ABB RobotStudio station: dual_weld_positioner.rspag

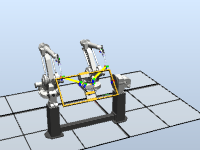
--- station ---
Station dual_weld_positioner (saved by RobotStudio 6.5.7392.129)
Controller 1410_dual_weld, task T_POS1: task frame (RAPID world) sits at (0, 0, 300) mm in the station
Controller 1410_dual_weld, task T_ROB2: task frame (RAPID world) sits at (0, 0, 300) mm in the station
Controller 1410_dual_weld, task T_ROB1: task frame (RAPID world) sits at (0, 0, 300) mm in the station
Controller 1410_dual_weld
  mechanical unit ROB_1: IRB1410_5_144__01, 6 joints, base frame (0, 0, 0) mm
  mechanical unit ROB_2: IRB1410_5_144__01_2, 6 joints, base frame (0, -1088.08, 0) mm
  mechanical unit STN1: IRBP_L300_L1250_M2009_REV1_01, 1 joints, base frame (1232.35, 0, 650) mm, rotated rx 0 ry -90 rz 90 deg
Layout (positions relative to the parent item):
  - IRB1410_5_144__01 [mechanism, from Robots\IRB1410_5_144_G_01.rslib] at (0, 0, 300) mm; joint values [0, -0.6808, -0.1899, 0, 0.7135, 0] (rad or m)
  - IRB1410_5_144__01_2 [mechanism, from Robots\IRB1410_5_144_G_01.rslib] at (0, -1088.08, 300) mm; joint values [0, -0.4622, -0.0882, 0, 0.6118, 0] (rad or m)
  - IRBP_L300_L1250_M2009_REV1_01 [mechanism] at (1232.35, 0, 0) mm; joint values [-0.7854] (rad or m)
      links: Base, Link1
  - test part [part] at (1232.35, 0, 950) mm, rotated rx 90 ry -45 rz 0 deg
  - Binzel_air_22 [mechanism, from Tools\Binzel_air_22.rslib] at (530.37, 0, 1452.5) mm, rotated rx 180 ry 60 rz 180 deg
  - Binzel_air_22_2 [mechanism, from Tools\Binzel_air_22.rslib] at (662.71, -1088.08, 1452.5) mm, rotated rx -180 ry 60 rz -180 deg
Attachment: test part is attached to IRBP_L300_L1250_M2009_REV1_01 / Link1
Attachment: Binzel_air_22 is attached to IRB1410_5_144__01 / Link6
Attachment: Binzel_air_22_2 is attached to IRB1410_5_144__01_2 / Link6

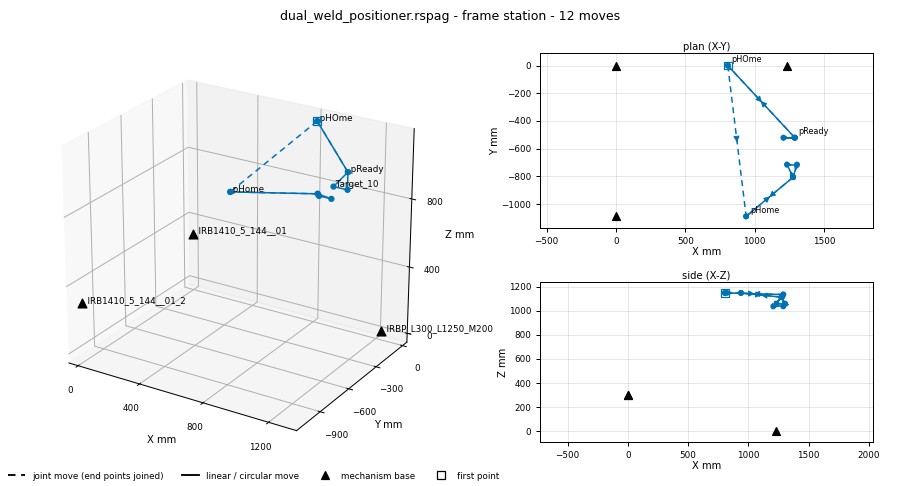
[picture p0: tool path of dual_weld_positioner.rspag in frame station, 12 of 17 moves have a stored position in this frame; points joined in program order, loops and branches not executed]
--- Backups/1410_dual_weld/RAPID/TASK1/PROGMOD/CalibData.mod ---
MODULE CalibData
	PERS tooldata tWeldGun:=[TRUE,[[125.800591275,0,391.268161315],[0.898794046,0,0.438371147,0]],[3,[0,0,100],[0,1,0,0],0,0,0]];
ENDMODULE

--- Backups/1410_dual_weld/RAPID/TASK1/PROGMOD/Module1.mod ---
MODULE Module1
    CONST robtarget pHOme:=[[806.318054074,0,847.919423179],[0.069756481,0,0.99756405,0],[0,0,0,0],[9E+09,9E+09,9E+09,9E+09,9E+09,9E+09]];
    CONST robtarget pReady:=[[1289.982978993,-520.829920074,834.561570832],[0.069756682,-0.00000004,0.997564036,-0.000000048],[-1,0,-1,0],[9E+09,9E+09,9E+09,9E+09,9E+09,9E+09]];
    CONST robtarget Target_10:=[[1207.204988688,-520.829978488,736.805052893],[0.06975661,-0.000000027,0.997564041,-0.000000051],[-1,0,-1,0],[9E+09,9E+09,9E+09,9E+09,9E+09,9E+09]];
    CONST robtarget Target_20:=[[1289.98298789,-520.829945867,736.805062664],[0.06975665,-0.000000033,0.997564038,-0.000000053],[-1,0,-1,0],[9E+09,9E+09,9E+09,9E+09,9E+09,9E+09]];
    VAR syncident sync1;
    VAR syncident sync2;
    VAR syncident sync3;
    VAR syncident sync4;
    PERS tasks all_tasks{3}:=[["T_ROB1"],["T_ROB2"],["T_POS1"]];

    PROC Path_10()
        MoveJ pHOme,v1000,fine,tWeldGun\WObj:=wobj0;
        WaitSyncTask sync1,all_tasks;
        MoveL pReady,v1000,fine,tWeldGun\WObj:=wobj0;
        MoveL Target_10,v1000,fine,tWeldGun\WObj:=wobj0;
        MoveL Target_20,v50,fine,tWeldGun\WObj:=wobj0;
        MoveL pReady,v1000,fine,tWeldGun\WObj:=wobj0;
        WaitSyncTask sync2,all_tasks;
        WaitSyncTask sync3,all_tasks;
        MoveJ pHOme,v1000,fine,tWeldGun\WObj:=wobj0;
        WaitSyncTask sync4,all_tasks;
    ENDPROC

    PROC main()
        Path_10;
    ENDPROC
ENDMODULE

--- Backups/1410_dual_weld/RAPID/TASK1/SYSMOD/LINKEDM.sys ---
%%%
  VERSION:1
  LANGUAGE:ENGLISH
%%%

MODULE LINKEDM (SYSMODULE)

! FOLLOWER
!     Name of electronically linked follower axis used by operator at teach pendent.
      PERS string l_f_axis_name{5}       :=  ["",  "", "", "", ""];

!     Name of the mechanical unit for follower axis.
      PERS string l_f_mecunt_n{5}  :=  ["", "", "", "", ""];

!     Linked follower axis number in the mechanical unit (first axis in mech. unit is number 1).
      PERS num l_f_axis_no{5}      :=  [0,          0,   0,  0,  0];

! MASTER
!     Name of the mechanical unit for linked master axis.
      PERS string l_m_mecunt_n{5} :=  ["", "", "", "", ""];

!     Linked master axis number in the mechanical unit (first axis in mech. unit is number 1).
!     See axis number table in documentation for different master mechanical units.
      PERS num l_m_axis_no{5}     :=  [0,  0,  0,  0,  0];

! POSITION OFFSET
!     The increase of the allowed offset position between the master and follower
!     positions, used when starting AUTO mode. As soon as the offset is decreased
!     the old configurated parameter is used.
!     Example: 3 => the configurated value of allowed offset is increased 3 times.
      PERS num offset_ratio{5}       :=  [10,  10,   10,  10,  10];

! SPEED RATIO
!     Speed_ratio used in AUTO and JOG modes [ very_slow   slow    normal    fast]
!     Value 1 = max allowed manual speed.
      CONST num speed_ratio {20}      := [0.01, 0.01, 0.01, 0.01, 0.01,
                                          0.05, 0.05, 0.05, 0.05, 0.05,
                                          0.20, 0.20, 0.20, 0.20, 0.20,
                                          1.00, 1.00, 1.00, 1.00, 1.00];

! STEP SIZE
!     Displacement position used in JOG mode for each activation of positive or
!     negative movement.                  [very_short    short   normal   long]
!     Unit degees or meter.
      CONST num displacement {20}     := [0.001, 0.001, 0.001, 0.001, 0.001,
                                          0.005, 0.005, 0.005, 0.005, 0.005,
                                          0.020, 0.020, 0.020, 0.020, 0.020,
                                          0.100, 0.100, 0.100, 0.100, 0.100];


!-------------------------------------------------------------
 PROC Linked_m ()
      Linked_m_exe ;
 ENDPROC
ENDMODULE

--- Backups/1410_dual_weld/RAPID/TASK2/PROGMOD/Module1.mod ---
MODULE Module1
	CONST robtarget pHome:=[[938.654977018,-1088.083832521,847.919435694],[0.0697565,0,0.997564048,0],[0,-1,0,0],[9E+09,9E+09,9E+09,9E+09,9E+09,9E+09]];
	CONST robtarget pReady:=[[1277.525959151,-805.567144457,812.597612335],[0.069756663,-0.000000019,0.997564037,0.000000002],[0,-1,0,0],[9E+09,9E+09,9E+09,9E+09,9E+09,9E+09]];
	CONST robtarget Target_10:=[[1233.430932885,-714.578767722,759.166040843],[0.069756556,0.000000008,0.997564045,0.000000014],[0,-1,0,0],[9E+09,9E+09,9E+09,9E+09,9E+09,9E+09]];
	CONST robtarget Target_20:=[[1305.430939185,-714.57875353,759.166041423],[0.069756582,-0.000000002,0.997564043,0.000000003],[0,-1,0,0],[9E+09,9E+09,9E+09,9E+09,9E+09,9E+09]];
	VAR syncident sync1;
    VAR syncident sync2;
    VAR syncident sync3;
    VAR syncident sync4;
    PERS tasks all_tasks{3}:=[["T_ROB1"],["T_ROB2"],["T_POS1"]];
    PROC Path_10()
	    MoveJ pHome,v1000,z100,tWeldGun\WObj:=wobj0;
           WaitSyncTask sync1,all_tasks;
	    MoveL pReady,v1000,z100,tWeldGun\WObj:=wobj0;
           WaitSyncTask sync2,all_tasks;
	    MoveL Target_10,v1000,z100,tWeldGun\WObj:=wobj0;
	    MoveL Target_20,v50,z100,tWeldGun\WObj:=wobj0;
         MoveL pReady,v1000,fine,tWeldGun\WObj:=wobj0;
        WaitSyncTask sync3,all_tasks;
        MoveJ pHome,v1000,z100,tWeldGun\WObj:=wobj0;
        WaitSyncTask sync4,all_tasks;
	ENDPROC
	PROC main()
	    Path_10;
	ENDPROC
ENDMODULE

--- Backups/1410_dual_weld/RAPID/TASK3/PROGMOD/Module1.mod ---
MODULE Module1
	CONST jointtarget pHome:=[[0,0,0,0,0,0],[9E+09,9E+09,9E+09,9E+09,-45,9E+09]];
	CONST jointtarget pWork:=[[0,0,0,0,0,0],[9E+09,9E+09,9E+09,9E+09,0,9E+09]];
    VAR syncident sync1;
VAR syncident sync2;
VAR syncident sync3;
VAR syncident sync4;
PERS tasks all_tasks{3} := [["T_ROB1"],["T_ROB2"],["T_POS1"]];


	PROC Path_10()
        ActUnit STN1;
	    MoveExtJ pHome,vrot50,fine;
	    MoveExtJ pWork,vrot50,fine;
        WaitSyncTask sync1,all_tasks;
        WaitSyncTask sync2,all_tasks;
          WaitSyncTask sync3,all_tasks;
          WaitSyncTask sync4,all_tasks;
          MoveExtJ pHome,vrot50,fine;
	ENDPROC
	PROC main()
	    Path_10;
	ENDPROC
    PROC Path_20()
        MoveExtJ pHome,vrot50,fine;
        MoveExtJ pWork,vrot50,fine;
    ENDPROC
ENDMODULE

--- Backups/1410_dual_weld/SYSPAR/EIO.cfg ---
EIO:CFG_1.0:6:1::
#
LOCAL_DEVICE:

      -Name "DRVIO_1" -Network "Local" -StateWhenStartup "Deactivated"\
      -TrustLevel "DRVIO_TRUSTLEVEL"
#
EIO_CROSS:

      -Name "Cross_doACT_K1" -Res "doACT_K1" -Act1 "soACT_STN1"

      -Name "Cross_siSTN1_ACT" -Res "siSTN1_ACT" -Act1 "diK1_ACT"
#
EIO_DEVICE_TRUSTLEVEL:

      -Name "DRVIO_TRUSTLEVEL" -ActionWhenLost "NONE" -ReportWhenLost "NONE"\
      -ReportWhenReconnected "NONE"
#
EIO_SIGNAL:

      -Name "doACT_K1" -SignalType "DO" -Device "DRVIO_1" -DeviceMap "0"

      -Name "doACT_K11" -SignalType "DO" -Device "DRVIO_1" -DeviceMap "5"

      -Name "diK1_ACT" -SignalType "DI" -Device "DRVIO_1" -DeviceMap "0"\
      -FiltPas 50 -FiltAct 50

      -Name "soACT_STN1" -SignalType "DO" -DeviceMap "0"

      -Name "siSTN1_ACT" -SignalType "DI" -DeviceMap "0"
